{attribute 'GeneratedUsingTerminal: EL5152-0000-0018'}
{attribute addProperty BoxType "EL5152-0000-0018"}
{attribute addProperty Id "StatusAT %I*Status_56494C1D6Counter_valueAT %I*UINT2"}
{attribute addProperty CRC "4194454294"}
{attribute addProperty Size "8"}
TYPE ENC_Status_compact_Channel_FA024B16 :
STRUCT
	{attribute addProperty Name "Status"}
	Status AT %I* : Status_56494C1D;
	{attribute addProperty Name "Counter_value"}
	Counter_value AT %I* : UINT;
END_STRUCT
END_TYPE

(* stored: Version 1.2.0.0, ProductVersion 3.1.4024.9
   DUT ENC_Status_compact_Channel_FA024B16: Id {7ade8572-2e40-49ce-9b04-7b4501b7fa95} *)
